KUKA KRL program: points1.src, points1.dat

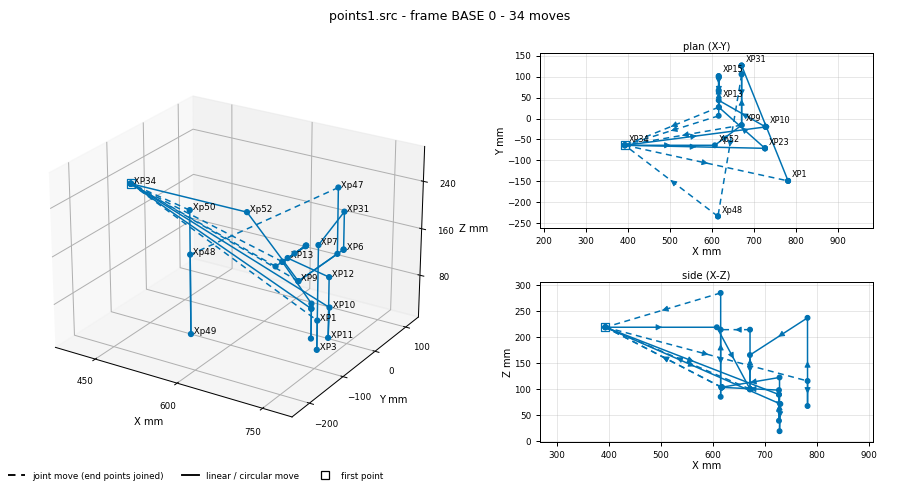
[picture p0: tool path of points1.src in frame BASE 0, 34 of 35 moves have a stored position in this frame; points joined in program order, loops and branches not executed]
--- points1.src ---
&ACCESS RVP
&REL 695
&PARAM TEMPLATE = C:\KRC\Roboter\Template\vorgabe
&PARAM EDITMASK = *
DEF points1( )
;FOLD INI
  ;FOLD BASISTECH INI
    GLOBAL INTERRUPT DECL 3 WHEN $STOPMESS==TRUE DO IR_STOPM ( )
    INTERRUPT ON 3
    BAS (#INITMOV,0 )
  ;ENDFOLD (BASISTECH INI)
  ;FOLD USER INI
    ;Make your modifications here

  ;ENDFOLD (USER INI)
;ENDFOLD (INI)


;FOLD PTP HOME Vel=100 % DEFAULT;%{PE}%R 5.6.11,%MKUKATPBASIS,%CMOVE,%VPTP,%P 1:PTP, 2:HOME, 3:, 5:100, 7:DEFAULT
$BWDSTART=FALSE
PDAT_ACT=PDEFAULT
FDAT_ACT=FHOME
BAS(#PTP_PARAMS,100)
$H_POS=XHOME
PTP XHOME
;ENDFOLD

;;goto wait postion
;FOLD PTP P34 Vel=100 % PDAT15 Tool[4]:Pneumatic_gripper Base[0];%{PE}%R 5.6.11,%MKUKATPBASIS,%CMOVE,%VPTP,%P 1:PTP, 2:P34, 3:, 5:100, 7:PDAT15
$BWDSTART=FALSE
PDAT_ACT=PPDAT15
FDAT_ACT=FP34
BAS(#PTP_PARAMS,100)
PTP XP34
;ENDFOLD

;;P1 approach
;FOLD PTP P1 CONT Vel=100 % PDAT1 Tool[4]:Pneumatic_gripper Base[0];%{PE}%R 5.6.11,%MKUKATPBASIS,%CMOVE,%VPTP,%P 1:PTP, 2:P1, 3:C_PTP, 5:100, 7:PDAT1
$BWDSTART=FALSE
PDAT_ACT=PPDAT1
FDAT_ACT=FP1
BAS(#PTP_PARAMS,100)
PTP XP1 C_PTP
;ENDFOLD


;;open gripper
;FOLD OUT 1 'AB_OUT_0' State=TRUE ;%{PE}%R 5.6.11,%MKUKATPBASIS,%COUT,%VOUTX,%P 2:1, 3:AB_OUT_0, 5:TRUE, 6:
$OUT[1]=TRUE
;ENDFOLD


;FOLD WAIT Time=1 sec;%{PE}%R 5.6.11,%MKUKATPBASIS,%CWAIT,%VWAIT,%P 2:1
WAIT SEC 1
;ENDFOLD

;;P1 acqire
;FOLD LIN P3 Vel=2 m/s CPDAT1 Tool[4]:Pneumatic_gripper Base[0];%{PE}%R 5.6.11,%MKUKATPBASIS,%CMOVE,%VLIN,%P 1:LIN, 2:P3, 3:, 5:2, 7:CPDAT1
$BWDSTART=FALSE
LDAT_ACT=LCPDAT1
FDAT_ACT=FP3
BAS(#CP_PARAMS,2)
LIN XP3
;ENDFOLD


;;close gripper
;FOLD OUT 1 'AB_OUT_0' State=FALSE ;%{PE}%R 5.6.11,%MKUKATPBASIS,%COUT,%VOUTX,%P 2:1, 3:AB_OUT_0, 5:FALSE, 6:
$OUT[1]=FALSE
;ENDFOLD


;FOLD WAIT Time=1 sec;%{PE}%R 5.6.11,%MKUKATPBASIS,%CWAIT,%VWAIT,%P 2:1
WAIT SEC 1
;ENDFOLD


;;intermediate path pos to insert part1

;;P1 retract
;FOLD LIN P7 Vel=2 m/s CPDAT4 Tool[4]:Pneumatic_gripper Base[0];%{PE}%R 5.6.11,%MKUKATPBASIS,%CMOVE,%VLIN,%P 1:LIN, 2:P7, 3:, 5:2, 7:CPDAT4
$BWDSTART=FALSE
LDAT_ACT=LCPDAT4
FDAT_ACT=FP7
BAS(#CP_PARAMS,2)
LIN XP7
;ENDFOLD

;;P1 to Fix empty approach
;FOLD LIN P31 Vel=2 m/s CPDAT27 Tool[4]:Pneumatic_gripper Base[0];%{PE}%R 5.6.11,%MKUKATPBASIS,%CMOVE,%VLIN,%P 1:LIN, 2:P31, 3:, 5:2, 7:CPDAT27
$BWDSTART=FALSE
LDAT_ACT=LCPDAT27
FDAT_ACT=FP31
BAS(#CP_PARAMS,2)
LIN XP31
;ENDFOLD

;;insert P1 into Fix
;FOLD LIN P6 Vel=0.5 m/s CPDAT3 Tool[4]:Pneumatic_gripper Base[0];%{PE}%R 5.6.11,%MKUKATPBASIS,%CMOVE,%VLIN,%P 1:LIN, 2:P6, 3:, 5:0.5, 7:CPDAT3
$BWDSTART=FALSE
LDAT_ACT=LCPDAT3
FDAT_ACT=FP6
BAS(#CP_PARAMS,0.5)
LIN XP6
;ENDFOLD

;;open gripper
;FOLD OUT 1 'AB_OUT_0' State=TRUE ;%{PE}%R 5.6.11,%MKUKATPBASIS,%COUT,%VOUTX,%P 2:1, 3:AB_OUT_0, 5:TRUE, 6:
$OUT[1]=TRUE
;ENDFOLD


;FOLD WAIT Time=1 sec;%{PE}%R 5.6.11,%MKUKATPBASIS,%CWAIT,%VWAIT,%P 2:1
WAIT SEC 1
;ENDFOLD


;;retract from Fix
;FOLD LIN P8 Vel=0.5 m/s CPDAT5 Tool[4]:Pneumatic_gripper Base[0];%{PE}%R 5.6.11,%MKUKATPBASIS,%CMOVE,%VLIN,%P 1:LIN, 2:P8, 3:, 5:0.5, 7:CPDAT5
$BWDSTART=FALSE
LDAT_ACT=LCPDAT5
FDAT_ACT=FP8
BAS(#CP_PARAMS,0.5)
LIN XP8
;ENDFOLD


;FOLD LIN P9 Vel=0.5 m/s CPDAT6 Tool[4]:Pneumatic_gripper Base[0];%{PE}%R 5.6.11,%MKUKATPBASIS,%CMOVE,%VLIN,%P 1:LIN, 2:P9, 3:, 5:0.5, 7:CPDAT6
$BWDSTART=FALSE
LDAT_ACT=LCPDAT6
FDAT_ACT=FP9
BAS(#CP_PARAMS,0.5)
LIN XP9
;ENDFOLD


;;goto wait pos
;FOLD PTP p42 Vel=100 % PDAT18 Tool[4]:Pneumatic_gripper Base[0];%{PE}%R 5.6.11,%MKUKATPBASIS,%CMOVE,%VPTP,%P 1:PTP, 2:p42, 3:, 5:100, 7:PDAT18
$BWDSTART=FALSE
PDAT_ACT=PPDAT18
FDAT_ACT=Fp42
BAS(#PTP_PARAMS,100)
PTP Xp42
;ENDFOLD

;;P2P3 approach
;FOLD LIN P10 Vel=2 m/s CPDAT23 Tool[4]:Pneumatic_gripper Base[0];%{PE}%R 5.6.11,%MKUKATPBASIS,%CMOVE,%VLIN,%P 1:LIN, 2:P10, 3:, 5:2, 7:CPDAT23
$BWDSTART=FALSE
LDAT_ACT=LCPDAT23
FDAT_ACT=FP10
BAS(#CP_PARAMS,2)
LIN XP10
;ENDFOLD

;;open gripper

;FOLD OUT 1 'AB_OUT_0' State=TRUE CONT;%{PE}%R 5.6.11,%MKUKATPBASIS,%COUT,%VOUTX,%P 2:1, 3:AB_OUT_0, 5:TRUE, 6:CONTINUE
CONTINUE
$OUT[1]=TRUE
;ENDFOLD

;FOLD WAIT Time=1 sec;%{PE}%R 5.6.11,%MKUKATPBASIS,%CWAIT,%VWAIT,%P 2:1
WAIT SEC 1
;ENDFOLD

;;acquire P2P3
;FOLD LIN P11 Vel=2 m/s CPDAT7 Tool[4]:Pneumatic_gripper Base[0];%{PE}%R 5.6.11,%MKUKATPBASIS,%CMOVE,%VLIN,%P 1:LIN, 2:P11, 3:, 5:2, 7:CPDAT7
$BWDSTART=FALSE
LDAT_ACT=LCPDAT7
FDAT_ACT=FP11
BAS(#CP_PARAMS,2)
LIN XP11
;ENDFOLD

;;close gripper
;FOLD OUT 1 'AB_OUT_0' State=FALSE ;%{PE}%R 5.6.11,%MKUKATPBASIS,%COUT,%VOUTX,%P 2:1, 3:AB_OUT_0, 5:FALSE, 6:
$OUT[1]=FALSE
;ENDFOLD

;FOLD WAIT Time=1 sec;%{PE}%R 5.6.11,%MKUKATPBASIS,%CWAIT,%VWAIT,%P 2:1
WAIT SEC 1
;ENDFOLD

;;retract P2P3
;FOLD LIN P12 Vel=2 m/s CPDAT8 Tool[4]:Pneumatic_gripper Base[0];%{PE}%R 5.6.11,%MKUKATPBASIS,%CMOVE,%VLIN,%P 1:LIN, 2:P12, 3:, 5:2, 7:CPDAT8
$BWDSTART=FALSE
LDAT_ACT=LCPDAT8
FDAT_ACT=FP12
BAS(#CP_PARAMS,2)
LIN XP12
;ENDFOLD

;;P2P3 to Approach P1Fix
;FOLD LIN P13 Vel=2 m/s CPDAT24 Tool[4]:Pneumatic_gripper Base[0];%{PE}%R 5.6.11,%MKUKATPBASIS,%CMOVE,%VLIN,%P 1:LIN, 2:P13, 3:, 5:2, 7:CPDAT24
$BWDSTART=FALSE
LDAT_ACT=LCPDAT24
FDAT_ACT=FP13
BAS(#CP_PARAMS,2)
LIN XP13
;ENDFOLD

;;P2P3 insert into P1Fix
;FOLD LIN P15 Vel=2 m/s CPDAT10 Tool[4]:Pneumatic_gripper Base[0];%{PE}%R 5.6.11,%MKUKATPBASIS,%CMOVE,%VLIN,%P 1:LIN, 2:P15, 3:, 5:2, 7:CPDAT10
$BWDSTART=FALSE
LDAT_ACT=LCPDAT10
FDAT_ACT=FP15
BAS(#CP_PARAMS,2)
LIN XP15
;ENDFOLD

;;open gripper
;FOLD OUT 1 'AB_OUT_0' State=TRUE ;%{PE}%R 5.6.11,%MKUKATPBASIS,%COUT,%VOUTX,%P 2:1, 3:AB_OUT_0, 5:TRUE, 6:
$OUT[1]=TRUE
;ENDFOLD

;FOLD WAIT Time=1 sec;%{PE}%R 5.6.11,%MKUKATPBASIS,%CWAIT,%VWAIT,%P 2:1
WAIT SEC 1
;ENDFOLD

;;Retract from P1P2P3Fix
;FOLD LIN P16 Vel=2 m/s CPDAT11 Tool[4]:Pneumatic_gripper Base[0];%{PE}%R 5.6.11,%MKUKATPBASIS,%CMOVE,%VLIN,%P 1:LIN, 2:P16, 3:, 5:2, 7:CPDAT11
$BWDSTART=FALSE
LDAT_ACT=LCPDAT11
FDAT_ACT=FP16
BAS(#CP_PARAMS,2)
LIN XP16
;ENDFOLD

;;close gripper
;FOLD OUT 1 'AB_OUT_0' State=FALSE ;%{PE}%R 5.6.11,%MKUKATPBASIS,%COUT,%VOUTX,%P 2:1, 3:AB_OUT_0, 5:FALSE, 6:
$OUT[1]=FALSE
;ENDFOLD

;FOLD WAIT Time=1 sec;%{PE}%R 5.6.11,%MKUKATPBASIS,%CWAIT,%VWAIT,%P 2:1
WAIT SEC 1
;ENDFOLD

;;nudge P2P3 into P1Fix
;FOLD LIN P17 Vel=2 m/s CPDAT12 Tool[4]:Pneumatic_gripper Base[0];%{PE}%R 5.6.11,%MKUKATPBASIS,%CMOVE,%VLIN,%P 1:LIN, 2:P17, 3:, 5:2, 7:CPDAT12
$BWDSTART=FALSE
LDAT_ACT=LCPDAT12
FDAT_ACT=FP17
BAS(#CP_PARAMS,2)
LIN XP17
;ENDFOLD

;;retract post nudge
;FOLD LIN P18 Vel=2 m/s CPDAT13 Tool[4]:Pneumatic_gripper Base[0];%{PE}%R 5.6.11,%MKUKATPBASIS,%CMOVE,%VLIN,%P 1:LIN, 2:P18, 3:, 5:2, 7:CPDAT13
$BWDSTART=FALSE
LDAT_ACT=LCPDAT13
FDAT_ACT=FP18
BAS(#CP_PARAMS,2)
LIN XP18
;ENDFOLD

;;goto wait position
;FOLD PTP p43 Vel=100 % PDAT19 Tool[4]:Pneumatic_gripper Base[0];%{PE}%R 5.6.11,%MKUKATPBASIS,%CMOVE,%VPTP,%P 1:PTP, 2:p43, 3:, 5:100, 7:PDAT19
$BWDSTART=FALSE
PDAT_ACT=PPDAT19
FDAT_ACT=Fp43
BAS(#PTP_PARAMS,100)
PTP Xp43
;ENDFOLD

;;P4 approach
;FOLD LIN P23 Vel=2 m/s CPDAT25 Tool[4]:Pneumatic_gripper Base[0];%{PE}%R 5.6.11,%MKUKATPBASIS,%CMOVE,%VLIN,%P 1:LIN, 2:P23, 3:, 5:2, 7:CPDAT25
$BWDSTART=FALSE
LDAT_ACT=LCPDAT25
FDAT_ACT=FP23
BAS(#CP_PARAMS,2)
LIN XP23
;ENDFOLD

;;open gripper
;FOLD OUT 1 'AB_OUT_0' State=TRUE ;%{PE}%R 5.6.11,%MKUKATPBASIS,%COUT,%VOUTX,%P 2:1, 3:AB_OUT_0, 5:TRUE, 6:
$OUT[1]=TRUE
;ENDFOLD

;FOLD WAIT Time=1 sec;%{PE}%R 5.6.11,%MKUKATPBASIS,%CWAIT,%VWAIT,%P 2:1
WAIT SEC 1
;ENDFOLD

;;P4 acqire
;FOLD LIN P27 Vel=2 m/s CPDAT19 Tool[4]:Pneumatic_gripper Base[0];%{PE}%R 5.6.11,%MKUKATPBASIS,%CMOVE,%VLIN,%P 1:LIN, 2:P27, 3:, 5:2, 7:CPDAT19
$BWDSTART=FALSE
LDAT_ACT=LCPDAT19
FDAT_ACT=FP27
BAS(#CP_PARAMS,2)
LIN XP27
;ENDFOLD


;FOLD LIN P24 Vel=2 m/s CPDAT17 Tool[4]:Pneumatic_gripper Base[0];%{PE}%R 5.6.11,%MKUKATPBASIS,%CMOVE,%VLIN,%P 1:LIN, 2:P24, 3:, 5:2, 7:CPDAT17
$BWDSTART=FALSE
LDAT_ACT=LCPDAT17
FDAT_ACT=FP24
BAS(#CP_PARAMS,2)
LIN XP24
;ENDFOLD



;FOLD OUT 1 'AB_OUT_0' State=FALSE ;%{PE}%R 5.6.11,%MKUKATPBASIS,%COUT,%VOUTX,%P 2:1, 3:AB_OUT_0, 5:FALSE, 6:
$OUT[1]=FALSE
;ENDFOLD

;FOLD WAIT Time=1 sec;%{PE}%R 5.6.11,%MKUKATPBASIS,%CWAIT,%VWAIT,%P 2:1
WAIT SEC 1
;ENDFOLD

;FOLD LIN P25 Vel=2 m/s CPDAT18 Tool[4]:Pneumatic_gripper Base[0];%{PE}%R 5.6.11,%MKUKATPBASIS,%CMOVE,%VLIN,%P 1:LIN, 2:P25, 3:, 5:2, 7:CPDAT18
$BWDSTART=FALSE
LDAT_ACT=LCPDAT18
FDAT_ACT=FP25
BAS(#CP_PARAMS,2)
LIN XP25
;ENDFOLD



;;P4 to approach P1P2P3Fix
;FOLD LIN P28 Vel=2 m/s CPDAT20 Tool[4]:Pneumatic_gripper Base[0];%{PE}%R 5.6.11,%MKUKATPBASIS,%CMOVE,%VLIN,%P 1:LIN, 2:P28, 3:, 5:2, 7:CPDAT20
$BWDSTART=FALSE
LDAT_ACT=LCPDAT20
FDAT_ACT=FP28
BAS(#CP_PARAMS,2)
LIN XP28
;ENDFOLD

;;P4 insert into P1P2P3Fix
;FOLD LIN P32 Vel=2 m/s CPDAT28 Tool[4]:Pneumatic_gripper Base[0];%{PE}%R 5.6.11,%MKUKATPBASIS,%CMOVE,%VLIN,%P 1:LIN, 2:P32, 3:, 5:2, 7:CPDAT28
$BWDSTART=FALSE
LDAT_ACT=LCPDAT28
FDAT_ACT=FP32
BAS(#CP_PARAMS,2)
LIN XP32
;ENDFOLD

;; wait for peg insertion
;FOLD WAIT Time=5 sec;%{PE}%R 5.6.11,%MKUKATPBASIS,%CWAIT,%VWAIT,%P 2:5
WAIT SEC 5
;ENDFOLD

;;open gripper
;FOLD OUT 1 'AB_OUT_0' State=TRUE ;%{PE}%R 5.6.11,%MKUKATPBASIS,%COUT,%VOUTX,%P 2:1, 3:AB_OUT_0, 5:TRUE, 6:
$OUT[1]=TRUE
;ENDFOLD

;FOLD WAIT Time=1 sec;%{PE}%R 5.6.11,%MKUKATPBASIS,%CWAIT,%VWAIT,%P 2:1
WAIT SEC 1
;ENDFOLD

;;retract from P1P2P3P4P5Fix
;FOLD LIN P30 Vel=2 m/s CPDAT22 Tool[4]:Pneumatic_gripper Base[0];%{PE}%R 5.6.11,%MKUKATPBASIS,%CMOVE,%VLIN,%P 1:LIN, 2:P30, 3:, 5:2, 7:CPDAT22
$BWDSTART=FALSE
LDAT_ACT=LCPDAT22
FDAT_ACT=FP30
BAS(#CP_PARAMS,2)
LIN XP30
;ENDFOLD

;; goto wait position
;FOLD PTP p44 Vel=100 % PDAT20 Tool[4]:Pneumatic_gripper Base[0];%{PE}%R 5.6.11,%MKUKATPBASIS,%CMOVE,%VPTP,%P 1:PTP, 2:p44, 3:, 5:100, 7:PDAT20
$BWDSTART=FALSE
PDAT_ACT=PPDAT20
FDAT_ACT=Fp44
BAS(#PTP_PARAMS,100)
PTP Xp44
;ENDFOLD

;;remove assembly

;;approach


;FOLD LIN p52 Vel=2 m/s CPDAT45 Tool[4]:Pneumatic_gripper Base[0];%{PE}%R 5.6.11,%MKUKATPBASIS,%CMOVE,%VLIN,%P 1:LIN, 2:p52, 3:, 5:2, 7:CPDAT45
$BWDSTART=FALSE
LDAT_ACT=LCPDAT45
FDAT_ACT=Fp52
BAS(#CP_PARAMS,2)
LIN Xp52
;ENDFOLD

;FOLD LIN p45 Vel=2 m/s CPDAT39 Tool[4]:Pneumatic_gripper Base[0];%{PE}%R 5.6.11,%MKUKATPBASIS,%CMOVE,%VLIN,%P 1:LIN, 2:p45, 3:, 5:2, 7:CPDAT39
$BWDSTART=FALSE
LDAT_ACT=LCPDAT39
FDAT_ACT=Fp45
BAS(#CP_PARAMS,2)
LIN Xp45
;ENDFOLD

;;open gripper

;FOLD OUT 1 'AB_OUT_0' State=TRUE ;%{PE}%R 5.6.11,%MKUKATPBASIS,%COUT,%VOUTX,%P 2:1, 3:AB_OUT_0, 5:TRUE, 6:
$OUT[1]=TRUE
;ENDFOLD

;FOLD WAIT Time=1 sec;%{PE}%R 5.6.11,%MKUKATPBASIS,%CWAIT,%VWAIT,%P 2:1
WAIT SEC 1
;ENDFOLD

;;acuire
;FOLD LIN p46 Vel=2 m/s CPDAT40 Tool[4]:Pneumatic_gripper Base[0];%{PE}%R 5.6.11,%MKUKATPBASIS,%CMOVE,%VLIN,%P 1:LIN, 2:p46, 3:, 5:2, 7:CPDAT40
$BWDSTART=FALSE
LDAT_ACT=LCPDAT40
FDAT_ACT=Fp46
BAS(#CP_PARAMS,2)
LIN Xp46
;ENDFOLD

;;close gripper
;FOLD OUT 1 'AB_OUT_0' State=FALSE ;%{PE}%R 5.6.11,%MKUKATPBASIS,%COUT,%VOUTX,%P 2:1, 3:AB_OUT_0, 5:FALSE, 6:
$OUT[1]=FALSE
;ENDFOLD

;FOLD WAIT Time=1 sec;%{PE}%R 5.6.11,%MKUKATPBASIS,%CWAIT,%VWAIT,%P 2:1
WAIT SEC 1
;ENDFOLD

;;retract
;FOLD LIN p47 Vel=2 m/s CPDAT41 Tool[4]:Pneumatic_gripper Base[0];%{PE}%R 5.6.11,%MKUKATPBASIS,%CMOVE,%VLIN,%P 1:LIN, 2:p47, 3:, 5:2, 7:CPDAT41
$BWDSTART=FALSE
LDAT_ACT=LCPDAT41
FDAT_ACT=Fp47
BAS(#CP_PARAMS,2)
LIN Xp47
;ENDFOLD

;; put on table
;FOLD PTP p48 Vel=100 % PDAT23 Tool[4]:Pneumatic_gripper Base[0];%{PE}%R 5.6.11,%MKUKATPBASIS,%CMOVE,%VPTP,%P 1:PTP, 2:p48, 3:, 5:100, 7:PDAT23
$BWDSTART=FALSE
PDAT_ACT=PPDAT23
FDAT_ACT=Fp48
BAS(#PTP_PARAMS,100)
PTP Xp48
;ENDFOLD

;FOLD LIN p49 Vel=2 m/s CPDAT43 Tool[4]:Pneumatic_gripper Base[0];%{PE}%R 5.6.11,%MKUKATPBASIS,%CMOVE,%VLIN,%P 1:LIN, 2:p49, 3:, 5:2, 7:CPDAT43
$BWDSTART=FALSE
LDAT_ACT=LCPDAT43
FDAT_ACT=Fp49
BAS(#CP_PARAMS,2)
LIN Xp49
;ENDFOLD

;FOLD OUT 1 'AB_OUT_0' State=TRUE ;%{PE}%R 5.6.11,%MKUKATPBASIS,%COUT,%VOUTX,%P 2:1, 3:AB_OUT_0, 5:TRUE, 6:
$OUT[1]=TRUE
;ENDFOLD

;FOLD WAIT Time=1 sec;%{PE}%R 5.6.11,%MKUKATPBASIS,%CWAIT,%VWAIT,%P 2:1
WAIT SEC 1
;ENDFOLD

;FOLD LIN p50 Vel=2 m/s CPDAT44 Tool[4]:Pneumatic_gripper Base[0];%{PE}%R 5.6.11,%MKUKATPBASIS,%CMOVE,%VLIN,%P 1:LIN, 2:p50, 3:, 5:2, 7:CPDAT44
$BWDSTART=FALSE
LDAT_ACT=LCPDAT44
FDAT_ACT=Fp50
BAS(#CP_PARAMS,2)
LIN Xp50
;ENDFOLD

;;goto wait postion

;FOLD PTP p51 Vel=100 % PDAT21 Tool[4]:Pneumatic_gripper Base[0];%{PE}%R 5.6.11,%MKUKATPBASIS,%CMOVE,%VPTP,%P 1:PTP, 2:p51, 3:, 5:100, 7:PDAT21
$BWDSTART=FALSE
PDAT_ACT=PPDAT21
FDAT_ACT=Fp51
BAS(#PTP_PARAMS,100)
PTP Xp51
;ENDFOLD

END

--- points1.dat ---
&ACCESS RVP
&REL 695
&PARAM TEMPLATE = C:\KRC\Roboter\Template\vorgabe
&PARAM EDITMASK = *
DEFDAT  POINTS1
;FOLD EXTERNAL DECLARATIONS;%{PE}%MKUKATPBASIS,%CEXT,%VCOMMON,%P
;FOLD BASISTECH EXT;%{PE}%MKUKATPBASIS,%CEXT,%VEXT,%P
EXT  BAS (BAS_COMMAND  :IN,REAL  :IN )
DECL INT SUCCESS
;ENDFOLD (BASISTECH EXT)
;FOLD USER EXT;%{E}%MKUKATPUSER,%CEXT,%VEXT,%P
;Make here your modifications

;ENDFOLD (USER EXT)
;ENDFOLD (EXTERNAL DECLARATIONS)
DECL BASIS_SUGG_T LAST_BASIS={POINT1[] "p53                     ",POINT2[] "p53                     ",CP_PARAMS[] "CPDAT45                 ",PTP_PARAMS[] "PDAT22                  ",CONT[] "                        ",CP_VEL[] "2                       ",PTP_VEL[] "100                     ",SYNC_PARAMS[] "SYNCDAT                 ",SPL_NAME[] "S0                      "}
DECL E6POS XP1={X 781.937683,Y -148.693604,Z 115.996201,A -173.269196,B 85.7474976,C -172.932297,S 2,T 41,E1 52.0275688,E2 0.0,E3 0.0,E4 0.0,E5 0.0,E6 0.0}
DECL FDAT FP1={TOOL_NO 4,BASE_NO 0,IPO_FRAME #BASE,POINT2[] " ",TQ_STATE FALSE}
DECL PDAT PPDAT1={VEL 100.0,ACC 100.0,APO_DIST 100.0,APO_MODE #CPTP}
DECL E6POS XP2={X 608.038513,Y -146.810898,Z 158.508606,A -172.487198,B 85.7499695,C -171.708496,S 2,T 41,E1 51.3119888,E2 0.0,E3 0.0,E4 0.0,E5 0.0,E6 0.0}
DECL FDAT FP2={TOOL_NO 1,BASE_NO 0,IPO_FRAME #BASE,POINT2[] " ",TQ_STATE FALSE}
DECL PDAT PPDAT2={VEL 100.0,ACC 100.0,APO_DIST 100.0,APO_MODE #CPTP}
DECL E6POS XP3={X 781.879028,Y -148.680206,Z 67.8220291,A -91.7551804,B 88.887207,C -91.3954391,S 2,T 43,E1 52.0206108,E2 0.0,E3 0.0,E4 0.0,E5 0.0,E6 0.0}
DECL FDAT FP3={TOOL_NO 4,BASE_NO 0,IPO_FRAME #BASE,POINT2[] " ",TQ_STATE FALSE}
DECL PDAT PPDAT3={VEL 100.0,ACC 100.0,APO_DIST 100.0,APO_MODE #CPTP}
DECL LDAT LCPDAT1={VEL 2.0,ACC 100.0,APO_DIST 100.0,APO_FAC 50.0,ORI_TYP #VAR,CIRC_TYP #BASE,JERK_FAC 50.0,EXAX_IGN 0}
DECL E6POS XP4={X 781.860229,Y -148.670395,Z 335.817505,A -92.1957779,B 88.8889236,C -91.8362427,S 2,T 41,E1 52.0174713,E2 0.0,E3 0.0,E4 0.0,E5 0.0,E6 0.0}
DECL FDAT FP4={TOOL_NO 4,BASE_NO 0,IPO_FRAME #BASE,POINT2[] " ",TQ_STATE FALSE}
DECL PDAT PPDAT4={VEL 100.0,ACC 100.0,APO_DIST 100.0,APO_MODE #CPTP}
DECL LDAT LCPDAT2={VEL 2.0,ACC 100.0,APO_DIST 100.0,APO_FAC 50.0,ORI_TYP #VAR,CIRC_TYP #BASE,JERK_FAC 50.0,EXAX_IGN 0}
DECL E6POS XP5={X 593.572021,Y 197.058395,Z 357.939301,A -177.582397,B 3.68012309,C 178.633301,S 2,T 33,E1 104.687103,E2 0.0,E3 0.0,E4 0.0,E5 0.0,E6 0.0}
DECL FDAT FP5={TOOL_NO 4,BASE_NO 0,IPO_FRAME #BASE,POINT2[] " ",TQ_STATE FALSE}
DECL PDAT PPDAT5={VEL 100.0,ACC 100.0,APO_DIST 100.0,APO_MODE #CPTP}
DECL E6POS XP6={X 671.013672,Y 126.269302,Z 99.6653137,A 90.5218201,B -0.255784303,C 92.8177338,S 2,T 11,E1 69.8371964,E2 0.0,E3 0.0,E4 0.0,E5 0.0,E6 0.0}
DECL FDAT FP6={TOOL_NO 4,BASE_NO 0,IPO_FRAME #BASE,POINT2[] " ",TQ_STATE FALSE}
DECL LDAT LCPDAT3={VEL 2.0,ACC 100.0,APO_DIST 100.0,APO_FAC 50.0,ORI_TYP #VAR,CIRC_TYP #BASE,JERK_FAC 50.0,EXAX_IGN 0}
DECL E6POS XP7={X 781.793701,Y -148.505402,Z 237.527802,A -92.3370209,B 88.943718,C -91.9763412,S 2,T 41,E1 52.0281715,E2 0.0,E3 0.0,E4 0.0,E5 0.0,E6 0.0}
DECL FDAT FP7={TOOL_NO 4,BASE_NO 0,IPO_FRAME #BASE,POINT2[] " ",TQ_STATE FALSE}
DECL LDAT LCPDAT4={VEL 2.0,ACC 100.0,APO_DIST 100.0,APO_FAC 50.0,ORI_TYP #VAR,CIRC_TYP #BASE,JERK_FAC 50.0,EXAX_IGN 0}
DECL E6POS XP8={X 671.173889,Y 126.041199,Z 100.461403,A 90.5082321,B -0.235773906,C 92.8068771,S 2,T 11,E1 69.8400497,E2 0.0,E3 0.0,E4 0.0,E5 0.0,E6 0.0}
DECL FDAT FP8={TOOL_NO 4,BASE_NO 0,IPO_FRAME #BASE,POINT2[] " ",TQ_STATE FALSE}
DECL LDAT LCPDAT5={VEL 2.0,ACC 100.0,APO_DIST 100.0,APO_FAC 50.0,ORI_TYP #VAR,CIRC_TYP #BASE,JERK_FAC 50.0,EXAX_IGN 0}
DECL E6POS XP9={X 671.174683,Y -15.7710896,Z 100.439003,A 90.5119171,B -0.241815701,C 92.809227,S 2,T 11,E1 69.8396912,E2 0.0,E3 0.0,E4 0.0,E5 0.0,E6 0.0}
DECL FDAT FP9={TOOL_NO 4,BASE_NO 0,IPO_FRAME #BASE,POINT2[] " ",TQ_STATE FALSE}
DECL LDAT LCPDAT6={VEL 2.0,ACC 100.0,APO_DIST 100.0,APO_FAC 50.0,ORI_TYP #VAR,CIRC_TYP #BASE,JERK_FAC 50.0,EXAX_IGN 0}
DECL E6POS XP10={X 729.552307,Y -19.8836308,Z 71.7596664,A 90.5600281,B -0.430729508,C 179.166306,S 2,T 33,E1 69.8371964,E2 0.0,E3 0.0,E4 0.0,E5 0.0,E6 0.0}
DECL FDAT FP10={TOOL_NO 4,BASE_NO 0,IPO_FRAME #BASE,POINT2[] " ",TQ_STATE FALSE}
DECL PDAT PPDAT6={VEL 100.0,ACC 100.0,APO_DIST 100.0,APO_MODE #CPTP}
DECL E6POS XP11={X 728.009705,Y -19.8733406,Z 19.3545094,A 90.5571899,B -0.432887614,C 179.174805,S 2,T 33,E1 69.8364029,E2 0.0,E3 0.0,E4 0.0,E5 0.0,E6 0.0}
DECL FDAT FP11={TOOL_NO 4,BASE_NO 0,IPO_FRAME #BASE,POINT2[] " ",TQ_STATE FALSE}
DECL LDAT LCPDAT7={VEL 2.0,ACC 100.0,APO_DIST 100.0,APO_FAC 50.0,ORI_TYP #VAR,CIRC_TYP #BASE,JERK_FAC 50.0,EXAX_IGN 0}
DECL E6POS XP12={X 727.940613,Y -19.8757095,Z 122.788002,A 90.5628128,B -0.43260631,C 179.1922,S 2,T 33,E1 69.8355331,E2 0.0,E3 0.0,E4 0.0,E5 0.0,E6 0.0}
DECL FDAT FP12={TOOL_NO 4,BASE_NO 0,IPO_FRAME #BASE,POINT2[] " ",TQ_STATE FALSE}
DECL LDAT LCPDAT8={VEL 2.0,ACC 100.0,APO_DIST 100.0,APO_FAC 50.0,ORI_TYP #VAR,CIRC_TYP #BASE,JERK_FAC 50.0,EXAX_IGN 0}
DECL E6POS XP13={X 616.470825,Y 43.3666801,Z 103.913101,A 153.748901,B -89.1171265,C 116.634102,S 2,T 35,E1 88.9031677,E2 0.0,E3 0.0,E4 0.0,E5 0.0,E6 0.0}
DECL FDAT FP13={TOOL_NO 4,BASE_NO 0,IPO_FRAME #BASE,POINT2[] " ",TQ_STATE FALSE}
DECL PDAT PPDAT7={VEL 100.0,ACC 100.0,APO_DIST 100.0,APO_MODE #CPTP}
DECL E6POS XP14={X 671.17157,Y -15.7369404,Z 667.470398,A 90.5185089,B -0.251326412,C 92.8096619,S 2,T 1,E1 69.8382263,E2 0.0,E3 0.0,E4 0.0,E5 0.0,E6 0.0}
DECL FDAT FP14={TOOL_NO 4,BASE_NO 0,IPO_FRAME #BASE,POINT2[] " ",TQ_STATE FALSE}
DECL LDAT LCPDAT9={VEL 2.0,ACC 100.0,APO_DIST 100.0,APO_FAC 50.0,ORI_TYP #VAR,CIRC_TYP #BASE,JERK_FAC 50.0,EXAX_IGN 0}
DECL E6POS XP15={X 616.450928,Y 101.2061,Z 103.8694,A 153.753006,B -89.1228638,C 116.631401,S 2,T 35,E1 88.901329,E2 0.0,E3 0.0,E4 0.0,E5 0.0,E6 0.0}
DECL FDAT FP15={TOOL_NO 4,BASE_NO 0,IPO_FRAME #BASE,POINT2[] " ",TQ_STATE FALSE}
DECL LDAT LCPDAT10={VEL 2.0,ACC 100.0,APO_DIST 100.0,APO_FAC 50.0,ORI_TYP #VAR,CIRC_TYP #BASE,JERK_FAC 50.0,EXAX_IGN 0}
DECL E6POS XP16={X 616.469788,Y 64.5801315,Z 103.835197,A 153.830597,B -89.1224899,C 116.548203,S 2,T 35,E1 88.9005966,E2 0.0,E3 0.0,E4 0.0,E5 0.0,E6 0.0}
DECL FDAT FP16={TOOL_NO 4,BASE_NO 0,IPO_FRAME #BASE,POINT2[] " ",TQ_STATE FALSE}
DECL LDAT LCPDAT11={VEL 2.0,ACC 100.0,APO_DIST 100.0,APO_FAC 50.0,ORI_TYP #VAR,CIRC_TYP #BASE,JERK_FAC 50.0,EXAX_IGN 0}
DECL E6POS XP17={X 616.473328,Y 100.8078,Z 103.805801,A 153.687393,B -89.1277466,C 116.688797,S 2,T 35,E1 88.8997269,E2 0.0,E3 0.0,E4 0.0,E5 0.0,E6 0.0}
DECL FDAT FP17={TOOL_NO 4,BASE_NO 0,IPO_FRAME #BASE,POINT2[] " ",TQ_STATE FALSE}
DECL LDAT LCPDAT12={VEL 2.0,ACC 100.0,APO_DIST 100.0,APO_FAC 50.0,ORI_TYP #VAR,CIRC_TYP #BASE,JERK_FAC 50.0,EXAX_IGN 0}
DECL E6POS XP18={X 616.461609,Y 6.41949415,Z 103.736801,A 154.130798,B -89.1225281,C 116.244698,S 2,T 35,E1 88.8976669,E2 0.0,E3 0.0,E4 0.0,E5 0.0,E6 0.0}
DECL FDAT FP18={TOOL_NO 4,BASE_NO 0,IPO_FRAME #BASE,POINT2[] " ",TQ_STATE FALSE}
DECL LDAT LCPDAT13={VEL 2.0,ACC 100.0,APO_DIST 100.0,APO_FAC 50.0,ORI_TYP #VAR,CIRC_TYP #BASE,JERK_FAC 50.0,EXAX_IGN 0}
DECL E6POS XP19={X 616.24408,Y -13.7945499,Z 117.046402,A 90.8169632,B -0.481606811,C -178.347,S 2,T 33,E1 88.8416367,E2 0.0,E3 0.0,E4 0.0,E5 0.0,E6 0.0}
DECL FDAT FP19={TOOL_NO 4,BASE_NO 0,IPO_FRAME #BASE,POINT2[] " ",TQ_STATE FALSE}
DECL PDAT PPDAT8={VEL 100.0,ACC 100.0,APO_DIST 100.0,APO_MODE #CPTP}
DECL E6POS XP20={X 857.356201,Y -76.5598602,Z 144.570908,A 114.675301,B -88.7251663,C 64.0555191,S 6,T 51,E1 92.9424133,E2 0.0,E3 0.0,E4 0.0,E5 0.0,E6 0.0}
DECL FDAT FP20={TOOL_NO 4,BASE_NO 0,IPO_FRAME #BASE,POINT2[] " ",TQ_STATE FALSE}
DECL PDAT PPDAT9={VEL 100.0,ACC 100.0,APO_DIST 100.0,APO_MODE #CPTP}
DECL E6POS XP21={X 857.259521,Y -76.5114822,Z 82.950798,A 113.443497,B -88.7815018,C 65.2834473,S 6,T 51,E1 92.9380035,E2 0.0,E3 0.0,E4 0.0,E5 0.0,E6 0.0}
DECL FDAT FP21={TOOL_NO 4,BASE_NO 0,IPO_FRAME #BASE,POINT2[] " ",TQ_STATE FALSE}
DECL LDAT LCPDAT14={VEL 2.0,ACC 100.0,APO_DIST 100.0,APO_FAC 50.0,ORI_TYP #VAR,CIRC_TYP #BASE,JERK_FAC 50.0,EXAX_IGN 0}
DECL E6POS XP22={X 857.256226,Y -76.4992676,Z 151.363098,A 113.2472,B -88.7788086,C 65.4797592,S 6,T 51,E1 92.9366837,E2 0.0,E3 0.0,E4 0.0,E5 0.0,E6 0.0}
DECL FDAT FP22={TOOL_NO 4,BASE_NO 0,IPO_FRAME #BASE,POINT2[] " ",TQ_STATE FALSE}
DECL LDAT LCPDAT15={VEL 2.0,ACC 100.0,APO_DIST 100.0,APO_FAC 50.0,ORI_TYP #VAR,CIRC_TYP #BASE,JERK_FAC 50.0,EXAX_IGN 0}
DECL E6POS XP23={X 726.823608,Y -71.0332794,Z 89.8683395,A 90.8105698,B -0.481687605,C -179.617203,S 2,T 33,E1 88.8828812,E2 0.0,E3 0.0,E4 0.0,E5 0.0,E6 0.0}
DECL FDAT FP23={TOOL_NO 4,BASE_NO 0,IPO_FRAME #BASE,POINT2[] " ",TQ_STATE FALSE}
DECL PDAT PPDAT10={VEL 100.0,ACC 100.0,APO_DIST 100.0,APO_MODE #CPTP}
DECL PDAT PPDAT11={VEL 100.0,ACC 100.0,APO_DIST 100.0,APO_MODE #CPTP}
DECL LDAT LCPDAT16={VEL 2.0,ACC 100.0,APO_DIST 100.0,APO_FAC 50.0,ORI_TYP #VAR,CIRC_TYP #BASE,JERK_FAC 50.0,EXAX_IGN 0}
DECL E6POS XP24={X 726.889526,Y -71.0537186,Z 39.4063988,A 90.8084717,B -0.48196429,C -179.632599,S 2,T 35,E1 88.8852921,E2 0.0,E3 0.0,E4 0.0,E5 0.0,E6 0.0}
DECL FDAT FP24={TOOL_NO 4,BASE_NO 0,IPO_FRAME #BASE,POINT2[] " ",TQ_STATE FALSE}
DECL LDAT LCPDAT17={VEL 2.0,ACC 100.0,APO_DIST 100.0,APO_FAC 50.0,ORI_TYP #VAR,CIRC_TYP #BASE,JERK_FAC 50.0,EXAX_IGN 0}
DECL E6POS XP25={X 726.856018,Y -71.0557785,Z 98.4238281,A 90.812767,B -0.481319308,C -179.624893,S 2,T 33,E1 88.8841934,E2 0.0,E3 0.0,E4 0.0,E5 0.0,E6 0.0}
DECL FDAT FP25={TOOL_NO 4,BASE_NO 0,IPO_FRAME #BASE,POINT2[] " ",TQ_STATE FALSE}
DECL LDAT LCPDAT18={VEL 2.0,ACC 100.0,APO_DIST 100.0,APO_FAC 50.0,ORI_TYP #VAR,CIRC_TYP #BASE,JERK_FAC 50.0,EXAX_IGN 0}
DECL E6POS XP26={X 616.793213,Y 15.6807098,Z 103.898804,A 141.281693,B -88.9675827,C 129.099701,S 2,T 35,E1 88.8828125,E2 0.0,E3 0.0,E4 0.0,E5 0.0,E6 0.0}
DECL FDAT FP26={TOOL_NO 4,BASE_NO 0,IPO_FRAME #BASE,POINT2[] " ",TQ_STATE FALSE}
DECL PDAT PPDAT12={VEL 100.0,ACC 100.0,APO_DIST 100.0,APO_MODE #CPTP}
DECL E6POS XP27={X 726.861206,Y -71.0438766,Z 89.9028091,A 90.8060532,B -0.482477397,C -179.6259,S 2,T 33,E1 88.8839111,E2 0.0,E3 0.0,E4 0.0,E5 0.0,E6 0.0}
DECL FDAT FP27={TOOL_NO 4,BASE_NO 0,IPO_FRAME #BASE,POINT2[] " ",TQ_STATE FALSE}
DECL LDAT LCPDAT19={VEL 2.0,ACC 100.0,APO_DIST 100.0,APO_FAC 50.0,ORI_TYP #VAR,CIRC_TYP #BASE,JERK_FAC 50.0,EXAX_IGN 0}
DECL E6POS XP28={X 616.850708,Y 26.8417492,Z 103.723801,A 141.065201,B -88.9753189,C 129.291107,S 2,T 35,E1 88.8767166,E2 0.0,E3 0.0,E4 0.0,E5 0.0,E6 0.0}
DECL FDAT FP28={TOOL_NO 4,BASE_NO 0,IPO_FRAME #BASE,POINT2[] " ",TQ_STATE FALSE}
DECL LDAT LCPDAT20={VEL 2.0,ACC 100.0,APO_DIST 100.0,APO_FAC 50.0,ORI_TYP #VAR,CIRC_TYP #BASE,JERK_FAC 50.0,EXAX_IGN 0}
DECL E6POS XP29={X 616.806519,Y 97.9642181,Z 103.843697,A 141.194794,B -88.9706497,C 129.176407,S 2,T 35,E1 88.8805389,E2 0.0,E3 0.0,E4 0.0,E5 0.0,E6 0.0}
DECL FDAT FP29={TOOL_NO 4,BASE_NO 0,IPO_FRAME #BASE,POINT2[] " ",TQ_STATE FALSE}
DECL PDAT PPDAT13={VEL 100.0,ACC 100.0,APO_DIST 100.0,APO_MODE #CPTP}
DECL LDAT LCPDAT21={VEL 2.0,ACC 100.0,APO_DIST 100.0,APO_FAC 50.0,ORI_TYP #VAR,CIRC_TYP #BASE,JERK_FAC 50.0,EXAX_IGN 0}
DECL E6POS XP30={X 616.798279,Y 27.0879307,Z 103.797203,A 141.313797,B -88.9719925,C 129.058304,S 2,T 35,E1 88.8789063,E2 0.0,E3 0.0,E4 0.0,E5 0.0,E6 0.0}
DECL FDAT FP30={TOOL_NO 4,BASE_NO 0,IPO_FRAME #BASE,POINT2[] " ",TQ_STATE FALSE}
DECL PDAT PPDAT14={VEL 100.0,ACC 100.0,APO_DIST 100.0,APO_MODE #CPTP}
DECL LDAT LCPDAT22={VEL 2.0,ACC 100.0,APO_DIST 100.0,APO_FAC 50.0,ORI_TYP #VAR,CIRC_TYP #BASE,JERK_FAC 50.0,EXAX_IGN 0}
DECL LDAT LCPDAT23={VEL 2.0,ACC 100.0,APO_DIST 100.0,APO_FAC 50.0,ORI_TYP #VAR,CIRC_TYP #BASE,JERK_FAC 50.0,EXAX_IGN 0}
DECL LDAT LCPDAT24={VEL 2.0,ACC 100.0,APO_DIST 100.0,APO_FAC 50.0,ORI_TYP #VAR,CIRC_TYP #BASE,JERK_FAC 50.0,EXAX_IGN 0}
DECL LDAT LCPDAT25={VEL 2.0,ACC 100.0,APO_DIST 100.0,APO_FAC 50.0,ORI_TYP #VAR,CIRC_TYP #BASE,JERK_FAC 50.0,EXAX_IGN 0}
DECL LDAT LCPDAT26={VEL 2.0,ACC 100.0,APO_DIST 100.0,APO_FAC 50.0,ORI_TYP #VAR,CIRC_TYP #BASE,JERK_FAC 50.0,EXAX_IGN 0}
DECL E6POS XP31={X 671.026001,Y 126.219902,Z 165.923401,A 90.5146027,B -0.250381887,C 92.8143692,S 2,T 11,E1 69.8382874,E2 0.0,E3 0.0,E4 0.0,E5 0.0,E6 0.0}
DECL FDAT FP31={TOOL_NO 4,BASE_NO 0,IPO_FRAME #BASE,POINT2[] " ",TQ_STATE FALSE}
DECL LDAT LCPDAT27={VEL 2.0,ACC 100.0,APO_DIST 100.0,APO_FAC 50.0,ORI_TYP #VAR,CIRC_TYP #BASE,JERK_FAC 50.0,EXAX_IGN 0}
DECL E6POS XP32={X 616.846375,Y 98.3731079,Z 103.726601,A 140.940201,B -88.9790268,C 129.409897,S 2,T 35,E1 88.8767929,E2 0.0,E3 0.0,E4 0.0,E5 0.0,E6 0.0}
DECL FDAT FP32={TOOL_NO 4,BASE_NO 0,IPO_FRAME #BASE,POINT2[] " ",TQ_STATE FALSE}
DECL LDAT LCPDAT28={VEL 2.0,ACC 100.0,APO_DIST 100.0,APO_FAC 50.0,ORI_TYP #VAR,CIRC_TYP #BASE,JERK_FAC 50.0,EXAX_IGN 0}
DECL E6POS XP33={X 392.891296,Y -63.8007011,Z 219.440598,A 1.80682504,B 1.23014903,C -179.629898,S 2,T 1,E1 88.8760071,E2 0.0,E3 0.0,E4 0.0,E5 0.0,E6 0.0}
DECL FDAT FP33={TOOL_NO 4,BASE_NO 0,IPO_FRAME #BASE,POINT2[] " ",TQ_STATE FALSE}
DECL LDAT LCPDAT29={VEL 2.0,ACC 100.0,APO_DIST 100.0,APO_FAC 50.0,ORI_TYP #VAR,CIRC_TYP #BASE,JERK_FAC 50.0,EXAX_IGN 0}
DECL E6POS XP34={X 392.871613,Y -63.8034706,Z 219.430496,A 1.80281198,B 1.23442996,C -179.630203,S 2,T 1,E1 88.8753967,E2 0.0,E3 0.0,E4 0.0,E5 0.0,E6 0.0}
DECL FDAT FP34={TOOL_NO 4,BASE_NO 0,IPO_FRAME #BASE,POINT2[] " ",TQ_STATE FALSE}
DECL LDAT LCPDAT30={VEL 2.0,ACC 100.0,APO_DIST 100.0,APO_FAC 50.0,ORI_TYP #VAR,CIRC_TYP #BASE,JERK_FAC 50.0,EXAX_IGN 0}
DECL PDAT PPDAT15={VEL 100.0,ACC 100.0,APO_DIST 100.0,APO_MODE #CPTP}
DECL E6POS XP35={X 616.820923,Y 75.1591797,Z 103.729698,A 141.124695,B -88.9779434,C 129.232407,S 2,T 35,E1 88.876358,E2 0.0,E3 0.0,E4 0.0,E5 0.0,E6 0.0}
DECL FDAT FP35={TOOL_NO 4,BASE_NO 0,IPO_FRAME #BASE,POINT2[] " ",TQ_STATE FALSE}
DECL LDAT LCPDAT31={VEL 2.0,ACC 100.0,APO_DIST 100.0,APO_FAC 50.0,ORI_TYP #VAR,CIRC_TYP #BASE,JERK_FAC 50.0,EXAX_IGN 0}
DECL E6POS XP36={X 616.832581,Y 36.4083214,Z 103.695702,A 141.191101,B -88.9776077,C 129.161804,S 2,T 35,E1 88.8753967,E2 0.0,E3 0.0,E4 0.0,E5 0.0,E6 0.0}
DECL FDAT FP36={TOOL_NO 4,BASE_NO 0,IPO_FRAME #BASE,POINT2[] " ",TQ_STATE FALSE}
DECL LDAT LCPDAT32={VEL 2.0,ACC 100.0,APO_DIST 100.0,APO_FAC 50.0,ORI_TYP #VAR,CIRC_TYP #BASE,JERK_FAC 50.0,EXAX_IGN 0}
DECL E6POS XP37={X 727.234497,Y 32.0601997,Z 26.5362206,A 90.5514908,B -0.441976696,C 179.174698,S 2,T 33,E1 69.8379364,E2 0.0,E3 0.0,E4 0.0,E5 0.0,E6 0.0}
DECL FDAT FP37={TOOL_NO 4,BASE_NO 0,IPO_FRAME #BASE,POINT2[] " ",TQ_STATE FALSE}
DECL LDAT LCPDAT33={VEL 2.0,ACC 100.0,APO_DIST 100.0,APO_FAC 50.0,ORI_TYP #VAR,CIRC_TYP #BASE,JERK_FAC 50.0,EXAX_IGN 0}
DECL E6POS XP38={X 727.255615,Y 32.0572395,Z 106.479401,A 90.5524063,B -0.442185313,C 179.1707,S 2,T 33,E1 69.8387375,E2 0.0,E3 0.0,E4 0.0,E5 0.0,E6 0.0}
DECL FDAT FP38={TOOL_NO 4,BASE_NO 0,IPO_FRAME #BASE,POINT2[] " ",TQ_STATE FALSE}
DECL LDAT LCPDAT34={VEL 2.0,ACC 100.0,APO_DIST 100.0,APO_FAC 50.0,ORI_TYP #VAR,CIRC_TYP #BASE,JERK_FAC 50.0,EXAX_IGN 0}
DECL E6POS XP39={X 613.910278,Y 129.317596,Z 122.622597,A 90.4514236,B -0.423337489,C 179.166107,S 2,T 33,E1 69.8366089,E2 0.0,E3 0.0,E4 0.0,E5 0.0,E6 0.0}
DECL FDAT FP39={TOOL_NO 4,BASE_NO 0,IPO_FRAME #BASE,POINT2[] " ",TQ_STATE FALSE}
DECL LDAT LCPDAT35={VEL 2.0,ACC 100.0,APO_DIST 100.0,APO_FAC 50.0,ORI_TYP #VAR,CIRC_TYP #BASE,JERK_FAC 50.0,EXAX_IGN 0}
DECL E6POS XP40={X 613.906921,Y 129.295395,Z 210.998596,A 90.4666138,B -0.4172768,C 179.168198,S 2,T 33,E1 69.8385773,E2 0.0,E3 0.0,E4 0.0,E5 0.0,E6 0.0}
DECL FDAT FP40={TOOL_NO 4,BASE_NO 0,IPO_FRAME #BASE,POINT2[] " ",TQ_STATE FALSE}
DECL LDAT LCPDAT36={VEL 2.0,ACC 100.0,APO_DIST 100.0,APO_FAC 50.0,ORI_TYP #VAR,CIRC_TYP #BASE,JERK_FAC 50.0,EXAX_IGN 0}
DECL E6POS XP41={X 613.906372,Y 129.295502,Z 210.998306,A 90.4666595,B -0.417255104,C 179.168198,S 2,T 33,E1 69.8385773,E2 0.0,E3 0.0,E4 0.0,E5 0.0,E6 0.0}
DECL FDAT FP41={TOOL_NO 4,BASE_NO 0,IPO_FRAME #BASE,POINT2[] " ",TQ_STATE FALSE}
DECL LDAT LCPDAT37={VEL 2.0,ACC 100.0,APO_DIST 100.0,APO_FAC 50.0,ORI_TYP #VAR,CIRC_TYP #BASE,JERK_FAC 50.0,EXAX_IGN 0}
DECL PDAT PPDAT16={VEL 100.0,ACC 100.0,APO_DIST 100.0,APO_MODE #CPTP}
DECL LDAT LCPDAT38={VEL 2.0,ACC 100.0,APO_DIST 100.0,APO_FAC 50.0,ORI_TYP #VAR,CIRC_TYP #BASE,JERK_FAC 50.0,EXAX_IGN 0}
DECL PDAT PPDAT17={VEL 100.0,ACC 100.0,APO_DIST 100.0,APO_MODE #CPTP}
DECL PDAT PPDAT18={VEL 100.0,ACC 100.0,APO_DIST 100.0,APO_MODE #CPTP}
DECL E6POS Xp42={X 392.871613,Y -63.8034706,Z 219.430496,A 1.80281198,B 1.23442996,C -179.630203,S 2,T 1,E1 88.8753967,E2 0.0,E3 0.0,E4 0.0,E5 0.0,E6 0.0}
DECL FDAT Fp42={TOOL_NO 4,BASE_NO 0,IPO_FRAME #BASE,POINT2[] " ",TQ_STATE FALSE}
DECL PDAT PPDAT19={VEL 100.0,ACC 100.0,APO_DIST 100.0,APO_MODE #CPTP}
DECL E6POS Xp43={X 392.871613,Y -63.8034706,Z 219.430496,A 1.80281198,B 1.23442996,C -179.630203,S 2,T 1,E1 88.8753967,E2 0.0,E3 0.0,E4 0.0,E5 0.0,E6 0.0}
DECL FDAT Fp43={TOOL_NO 4,BASE_NO 0,IPO_FRAME #BASE,POINT2[] " ",TQ_STATE FALSE}
DECL PDAT PPDAT20={VEL 100.0,ACC 100.0,APO_DIST 100.0,APO_MODE #CPTP}
DECL E6POS Xp44={X 392.871613,Y -63.8034706,Z 219.430496,A 1.80281198,B 1.23442996,C -179.630203,S 2,T 1,E1 88.8753967,E2 0.0,E3 0.0,E4 0.0,E5 0.0,E6 0.0}
DECL FDAT Fp44={TOOL_NO 4,BASE_NO 0,IPO_FRAME #BASE,POINT2[] " ",TQ_STATE FALSE}
DECL E6POS XP45={X 671.174683,Y -15.7612896,Z 100.427002,A 90.5131607,B -0.243338197,C 92.8100662,S 2,T 11,E1 69.8393936,E2 0.0,E3 0.0,E4 0.0,E5 0.0,E6 0.0}
DECL FDAT Fp45={TOOL_NO 4,BASE_NO 0,IPO_FRAME #BASE,POINT2[] " ",TQ_STATE FALSE}
DECL LDAT LCPDAT39={VEL 2.0,ACC 100.0,APO_DIST 100.0,APO_FAC 50.0,ORI_TYP #VAR,CIRC_TYP #BASE,JERK_FAC 50.0,EXAX_IGN 0}
DECL E6POS XP46={X 671.17157,Y 105.925102,Z 100.3834,A 90.5118179,B -0.239839897,C 92.8136597,S 2,T 11,E1 69.8383636,E2 0.0,E3 0.0,E4 0.0,E5 0.0,E6 0.0}
DECL FDAT Fp46={TOOL_NO 4,BASE_NO 0,IPO_FRAME #BASE,POINT2[] " ",TQ_STATE FALSE}
DECL LDAT LCPDAT40={VEL 2.0,ACC 100.0,APO_DIST 100.0,APO_FAC 50.0,ORI_TYP #VAR,CIRC_TYP #BASE,JERK_FAC 50.0,EXAX_IGN 0}
DECL E6POS XP47={X 671.174011,Y 104.913002,Z 214.754807,A 90.5100632,B -0.247895002,C 92.8193283,S 2,T 9,E1 69.835289,E2 0.0,E3 0.0,E4 0.0,E5 0.0,E6 0.0}
DECL FDAT Fp47={TOOL_NO 4,BASE_NO 0,IPO_FRAME #BASE,POINT2[] " ",TQ_STATE FALSE}
DECL LDAT LCPDAT41={VEL 2.0,ACC 100.0,APO_DIST 100.0,APO_FAC 50.0,ORI_TYP #VAR,CIRC_TYP #BASE,JERK_FAC 50.0,EXAX_IGN 0}
DECL E6POS XP48={X 614.69342,Y -233.138794,Z 214.795105,A -107.410698,B 88.3525009,C -104.551598,S 2,T 41,E1 69.8267975,E2 0.0,E3 0.0,E4 0.0,E5 0.0,E6 0.0}
DECL FDAT Fp48={TOOL_NO 4,BASE_NO 0,IPO_FRAME #BASE,POINT2[] " ",TQ_STATE FALSE}
DECL LDAT LCPDAT42={VEL 2.0,ACC 100.0,APO_DIST 100.0,APO_FAC 50.0,ORI_TYP #VAR,CIRC_TYP #BASE,JERK_FAC 50.0,EXAX_IGN 0}
DECL E6POS XP49={X 614.686584,Y -233.1492,Z 85.5402832,A -123.021599,B 89.0900879,C -120.163399,S 2,T 43,E1 69.8244629,E2 0.0,E3 0.0,E4 0.0,E5 0.0,E6 0.0}
DECL FDAT Fp49={TOOL_NO 4,BASE_NO 0,IPO_FRAME #BASE,POINT2[] " ",TQ_STATE FALSE}
DECL LDAT LCPDAT43={VEL 2.0,ACC 100.0,APO_DIST 100.0,APO_FAC 50.0,ORI_TYP #VAR,CIRC_TYP #BASE,JERK_FAC 50.0,EXAX_IGN 0}
DECL E6POS XP50={X 614.678223,Y -233.126404,Z 285.433014,A -107.671204,B 88.3475571,C -104.815102,S 2,T 41,E1 69.8240891,E2 0.0,E3 0.0,E4 0.0,E5 0.0,E6 0.0}
DECL FDAT Fp50={TOOL_NO 4,BASE_NO 0,IPO_FRAME #BASE,POINT2[] " ",TQ_STATE FALSE}
DECL LDAT LCPDAT44={VEL 2.0,ACC 100.0,APO_DIST 100.0,APO_FAC 50.0,ORI_TYP #VAR,CIRC_TYP #BASE,JERK_FAC 50.0,EXAX_IGN 0}
DECL PDAT PPDAT21={VEL 100.0,ACC 100.0,APO_DIST 100.0,APO_MODE #CPTP}
DECL E6POS Xp51={X 392.871613,Y -63.8034706,Z 219.430496,A 1.80281198,B 1.23442996,C -179.630203,S 2,T 1,E1 88.8753967,E2 0.0,E3 0.0,E4 0.0,E5 0.0,E6 0.0}
DECL FDAT Fp51={TOOL_NO 4,BASE_NO 0,IPO_FRAME #BASE,POINT2[] " ",TQ_STATE FALSE}
DECL E6POS XP52={X 607.299377,Y -63.7969589,Z 219.384705,A 1.80947495,B 1.238446,C -179.627106,S 2,T 1,E1 88.873497,E2 0.0,E3 0.0,E4 0.0,E5 0.0,E6 0.0}
DECL FDAT Fp52={TOOL_NO 4,BASE_NO 0,IPO_FRAME #BASE,POINT2[] " ",TQ_STATE FALSE}
DECL LDAT LCPDAT45={VEL 2.0,ACC 100.0,APO_DIST 100.0,APO_FAC 50.0,ORI_TYP #VAR,CIRC_TYP #BASE,JERK_FAC 50.0,EXAX_IGN 0}
DECL PDAT PPDAT22={VEL 100.0,ACC 100.0,APO_DIST 100.0,APO_MODE #CPTP}
DECL E6POS Xp53={X 392.871613,Y -63.8034706,Z 219.430496,A 1.80281198,B 1.23442996,C -179.630203,S 2,T 1,E1 88.8753967,E2 0.0,E3 0.0,E4 0.0,E5 0.0,E6 0.0}
DECL FDAT Fp53={TOOL_NO 4,BASE_NO 0,IPO_FRAME #BASE,POINT2[] " ",TQ_STATE FALSE}
DECL PDAT PPDAT23={VEL 100.0,ACC 100.0,APO_DIST 100.0,APO_MODE #CPTP}
ENDDAT
